Fanuc KAREL source: ko00004.KL

-- PROVISIONAL review KL for V940-1; original PC SHA256 fc5897f4519bbd870bbe302c28205e6281f1e44bd6826cff4be84b705553d7e1
-- Incomplete behavior may be omitted. Consult companion uncertainty JSON. Do not deploy.
PROGRAM KO00004
%NOLOCKGROUP
-- UNRESOLVED_DECL P1 type=000101
-- UNRESOLVED_DECL P2 type=000101
-- UNRESOLVED_DECL P3 type=000101
-- UNRESOLVED_DECL OUT type=000199
BEGIN
  -- V9_ZERO_TABLE_METADATA_HINT layout=0001; no indexed target words; source/name/runtime held
  -- UNRESOLVED_PC offsets 5-56; opcodes 27,22,1C,22,1C,22,1C,76,7E,4A
  -- UNRESOLVED_PC offsets 61-65; opcodes 7F
END KO00004
